TYPE ST_Bel_Stellwert :
STRUCT
	Betrieb					: BOOL;
	Freigabe_Stellwert		: BOOL;
	Leistung				: BYTE;
END_STRUCT
END_TYPE

(* stored: Version 1.1.0.1, ProductVersion 3.1.4024.9
   DUT ST_Bel_Stellwert: Id {803fd37f-3788-4a66-b2b8-78a46acaa6b2} *)
